FUNCTION_BLOCK CylinderLS (* Composite Function Block Type *)
  (* Standard: 61499-2 *)
  (* Version 0.0, 5/26/2016, Andrei, nxtControl GmbH, template *)
  PACKAGE Main;
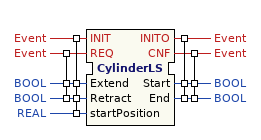
  EVENT_INPUT
    INIT WITH Extend, Retract, startPosition; (* Initialization Request *)
    REQ WITH Extend, Retract; (* Normal Execution Request *)
  END_EVENT
  EVENT_OUTPUT
    INITO WITH Start, End; (* Initialization Confirm *)
    CNF WITH Start, End; (* Execution Confirmation *)
  END_EVENT
  VAR_INPUT
    Extend : BOOL; (* Input event qualifier *)
    Retract : BOOL;
    startPosition : REAL;
  END_VAR
  VAR_OUTPUT
    Start : BOOL; (* Output event qualifier *)
    End : BOOL;
  END_VAR
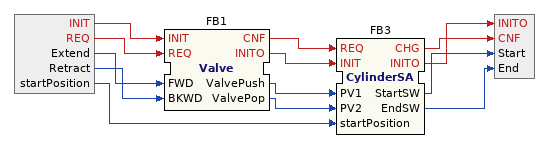
  FBS
    FB3 : CylinderSA;
    FB1 : Valve;
  END_FBS
  EVENT_CONNECTIONS
    FB3.CHG TO CNF;
    FB3.INITO TO INITO;
    FB1.CNF TO FB3.REQ;
    INIT TO FB1.INIT;
    REQ TO FB1.REQ;
    FB1.INITO TO FB3.INIT;
  END_CONNECTIONS
  DATA_CONNECTIONS
    FB3.StartSW TO Start;
    FB3.EndSW TO End;
    Extend TO FB1.FWD;
    Retract TO FB1.BKWD;
    FB1.ValvePush TO FB3.PV1;
    FB1.ValvePop TO FB3.PV2;
    startPosition TO FB3.startPosition;
  END_CONNECTIONS
END_FUNCTION_BLOCK
